TYPE Motion_Axis :
STRUCT
	AXIS 					: AXIS_REF;
	HOME_CALIBRATION AT %I* : BOOL;
END_STRUCT
END_TYPE

(* stored: Version 1.1.0.1, ProductVersion 3.1.0.36
   DUT Motion_Axis: Id {b6a92e77-5b6e-42e3-aa69-5b66e0d254e3} *)
